FUNCTION_BLOCK EM_LiftingTransport EXTENDS EM_Base IMPLEMENTS I_EM_LiftingTransport

VAR_INPUT
//Inputs
	i_ref_stSettings : REFERENCE TO ST_SettingsLiftingTransport;
	
	// External interlocks (from outside this EM)
	i_fbExtIlckLiftUp : FB_Interlock;
	i_fbExtIlckLiftDown : FB_Interlock;
	i_fbExtIlckTransportExtract : FB_Interlock;
	i_fbExtIlckTransportRetract : FB_Interlock;
	
	i_refTB : REFERENCE TO OBJ_Carrier;	//Mogelijk voor uiteindelijke machine, voor de FUMO's is dit nog niet echt relevant
	
	i_eCtrlState		: E_CtrlState;
	
	s_arr_bTest : ARRAY[0..15] OF BOOL; 
END_VAR

VAR_OUTPUT
	q_bStaWarning : BOOL;
END_VAR

VAR

	//Interlocks	
	fbIlckHandlerLiftUp : FB_InterlockHandler;
	fbIlckHandlerLiftDown : FB_InterlockHandler;

	fbIlckHandlerTransportExtract : FB_InterlockHandler;
	fbIlckHandlerTransportRetract : FB_InterlockHandler;

//------------------------------------------//
	//Control Modules (Devices)
	axisLift : AXIS_REF;
	s_cmLift : CM_AX5000; // Including 2 limit switched and 1 reference switch

	axisTransport : AXIS_REF;
	s_cmTransport : CM_AX5000; // Including 2 limit switched and 1 reference switch
	
//------------------------------------------//

//------------------------------------------//
//Inputs
	s_diStaTrolleyOnPositionLeft : FB_DigInput;
	s_diStaTrolleyOnPositionRight : FB_DigInput;
	s_diStaCabinAreaOccupied : FB_DigInput;
	s_diStaCollisionAvoidanceSensor : FB_DigInput;
	s_diStaTrolleyLocked : FB_DigInput;
	s_diStaTrolleyUnlocked : FB_DigInput;
//------------------------------------------//	
	
//------------------------------------------//
//Outputs

//------------------------------------------//

	//Requests
	s_bReqGoToIdle : BOOL := FALSE;
	s_bReqPickTrolleyFromTB : BOOL := FALSE;
	s_bReqPlaceTrolleyInTB : BOOL := FALSE;

	//States
	s_bStaLiftDriveError : BOOL := FALSE;
	s_bStaTransportDriveError : BOOL := FALSE;
	
	s_bStaTrolleyInCabin : BOOL := FALSE;
	s_bStaTrolleyInTB : BOOL := FALSE;
		
	s_bStaTrolleyOnPositionLeft : BOOL := FALSE;
	s_bStaTrolleyOnPositionRight : BOOL := FALSE;
	s_bStaCabinAreaOccupied : BOOL := FALSE;
	s_bStaCollisionAvoidanceSensor : BOOL := FALSE;
	s_bStaTrolleyLocked : BOOL := FALSE;
	s_bStaTrolleyUnlocked : BOOL := FALSE;
	
	//Properties
	s_bStaAtIdlePosition : BOOL := FALSE;
	s_bStaTrolleyPickedFromTB : BOOL := FALSE;
	s_bStaTrolleyPlacedInTB : BOOL := FALSE;	

	//Interlockes	
	s_bIlckLiftUp : BOOL := TRUE;
	s_bIlckLiftDown : BOOL := TRUE;
	s_bIlckTransportExtract : BOOL := TRUE;
	s_bIlckTransportRetract : BOOL := TRUE;
	
//Alarms
	s_sReason : STRING;
	
	s_fbAlarmHandlerLiftDrive : FB_AlarmHandler;
	s_fbAlarmHandlerTransportDrive : FB_AlarmHandler;
	
	s_bErrLiftDrive : BOOL;
	s_bErrTransportDrive : BOOL;
	
	//Warnings
	s_fbAlarmHandlerSafetyDoorNotClosed : FB_AlarmHandler;
	s_bWrnSafetyDoorNotClosed : BOOL;
	
	s_bStaWarning : BOOL;
	
	s_sMessage : STRING;

	//Sequencers
	s_eSeqLiftingTransport : E_SeqLiftingTransport;
	s_fbSeqLiftingTransportControl : FB_SeqControl;

	s_eTmpLocation : E_Location;
	s_eTmpCenteringDone : BOOL;
	
	s_tMaxTravelTime : TIME;
	s_tDoorCheckTime : TIME;
	s_bDoorCheckTimeDisabled : BOOL := FALSE;
	

	//Hmi
	//Buttons
	s_fbHmiBtnGoToIdle					: FB_HmiBtn;
	s_fbHmiBtnPickTrolleyFromTB			: FB_HmiBtn;
	s_fbHmiBtnPlaceTrolleyInTB			: FB_HmiBtn;
		
	//Leds
	s_fbHmiLedTrolleyOnPositionLeft		: FB_HmiLed;
	s_fbHmiLedTrolleyOnPositionRight	: FB_HmiLed;
	s_fbHmiLedCabinAreaOccupied			: FB_HmiLed;
	s_fbHmiLedCollisionAvoidanceSensor	: FB_HmiLed;
	s_fbHmiLedTrolleyLocked				: FB_HmiLed;
	s_fbHmiLedTrolleyUnlocked			: FB_HmiLed;
	
	{warning '#TODO' Het zou beter zijn om dit onder te brengen in de onderstaande control modules}
	s_bHmiForceOutputEnabled : BOOL;
END_VAR

	
SUPER^();

METHOD PROTECTED _m_Alarms : BOOL

IF NOT SUPER^._m_Alarms() THEN
	RETURN;
END_IF

// Alarm Handlers
s_fbAlarmHandlerLiftDrive(
	i_bStaActive := s_bErrLiftDrive, 
	i_eAlarmLevel := E_AlarmLevel.Alarm, 
	i_sAlarmText := CONCAT(i_sEmName, CONCAT( ': Scissor Lift Drive error: ', s_sReason)));
	
s_fbAlarmHandlerTransportDrive(
	i_bStaActive := s_bErrTransportDrive, 
	i_eAlarmLevel := E_AlarmLevel.Alarm, 
	i_sAlarmText := CONCAT(i_sEmName, CONCAT( ': Transport Unit Drive error: ', s_sReason)));

// Reset warnings
IF i_bCmdReset THEN
	s_bWrnSafetyDoorNotClosed := FALSE;
END_IF

s_bStaError := 
	s_cmLift.p_bError
	OR s_cmTransport.p_bError
	OR s_fbAlarmHandlerLiftDrive.q_bStaActive
	OR s_fbAlarmHandlerTransportDrive.q_bStaActive;
	
s_bStaWarning :=
	s_fbAlarmHandlerSafetyDoorNotClosed.q_bStaActive;
	
_m_Alarms := TRUE;
END_METHOD

METHOD PRIVATE _m_AutomaticControl : BOOL

//Lifting Transport
_m_SeqLiftingTransport();
END_METHOD

METHOD PROTECTED _m_Devices : BOOL

IF NOT SUPER^._m_Devices() THEN
	RETURN;
END_IF

s_cmLift(
	i_bReqEnable := i_bReqEnable,
	i_eCtrlMode := i_eCtrlMode,
	i_bCmdReset := i_bCmdReset,
	i_refAxis := axisLift,
	i_bIclkForward := s_bIlckLiftUp,
	i_bIclkBackward := s_bIlckLiftDown);

s_bStaLiftDriveError := s_cmLift.p_bError;
	
s_cmTransport(
	i_bReqEnable := i_bReqEnable,
	i_eCtrlMode := i_eCtrlMode,
	i_bCmdReset := i_bCmdReset,
	i_refAxis := axisTransport,
	i_bIclkForward := s_bIlckTransportExtract, 
	i_bIclkBackward := s_bIlckTransportRetract);

s_bStaTransportDriveError := s_cmTransport.p_bError;

s_diStaTrolleyOnPositionLeft();
s_diStaTrolleyOnPositionRight();
s_diStaCabinAreaOccupied();
s_diStaCollisionAvoidanceSensor();
s_diStaTrolleyLocked();
s_diStaTrolleyUnlocked();

s_bStaTrolleyOnPositionLeft := s_diStaTrolleyOnPositionLeft.p_bStaInputDelayed;
s_bStaTrolleyOnPositionRight := s_diStaTrolleyOnPositionRight.p_bStaInputDelayed;
s_bStaCabinAreaOccupied := s_diStaCabinAreaOccupied.p_bStaInputDelayed;
s_bStaCollisionAvoidanceSensor := s_diStaCollisionAvoidanceSensor.p_bStaInputDelayed;
s_bStaTrolleyLocked := s_diStaTrolleyLocked.p_bStaInputDelayed;
s_bStaTrolleyUnlocked := s_diStaTrolleyUnlocked.p_bStaInputDelayed;

_m_Devices := TRUE;
END_METHOD

METHOD PROTECTED _m_Hmi : BOOL

IF NOT SUPER^._m_Hmi() THEN
	RETURN;
END_IF

//Buttons
s_fbHmiBtnGoToIdle();
s_fbHmiBtnPickTrolleyFromTB();
s_fbHmiBtnPlaceTrolleyInTB();

//Leds

s_fbHmiLedTrolleyOnPositionLeft(i_bStaLed := s_bStaTrolleyOnPositionLeft);
s_fbHmiLedTrolleyOnPositionRight(i_bStaLed := s_bStaTrolleyOnPositionRight);
s_fbHmiLedCabinAreaOccupied(i_bStaLed := s_bStaCabinAreaOccupied);
s_fbHmiLedCollisionAvoidanceSensor(i_bStaLed := s_bStaCollisionAvoidanceSensor);
s_fbHmiLedTrolleyLocked(i_bStaLed := s_bStaTrolleyLocked);
s_fbHmiLedTrolleyUnlocked(i_bStaLed := s_bStaTrolleyUnlocked);

_m_Hmi := TRUE;
END_METHOD

METHOD PROTECTED _m_Init : BOOL

IF NOT SUPER^._m_Init() THEN
	RETURN;
END_IF

//Control Modules
s_cmLift.i_bReqEnable := FALSE;
s_cmLift.i_eCtrlMode := E_CtrlMode.IDLE;
s_cmLift.i_sCmName := 'CM Lift';
s_cmLift.i_refAxis REF= axisLift;

s_cmTransport.i_bReqEnable := FALSE;
s_cmTransport.i_eCtrlMode := E_CtrlMode.IDLE;
s_cmTransport.i_sCmName := 'CM Transport Unit';
s_cmTransport.i_refAxis REF= axisTransport;
{warning '#TODO: Dot we need to added configuration parameters? Seperate struct or via settings or dedicateed variables'}

s_diStaTrolleyOnPositionLeft.i_stSettings.tmInputDelay := T#100MS;
s_diStaTrolleyOnPositionRight.i_stSettings.tmInputDelay := T#100MS;
s_diStaCabinAreaOccupied.i_stSettings.tmInputDelay := T#100MS;
s_diStaCollisionAvoidanceSensor.i_stSettings.tmInputDelay := T#100MS;
s_diStaTrolleyLocked.i_stSettings.tmInputDelay := T#100MS;
s_diStaTrolleyUnlocked.i_stSettings.tmInputDelay := T#100MS;

//Interlock strings
//Lift
//	i_stInterlockList.arr_Interlocks[0].sReason --> External, dynamical will be written in m_input
	fbIlckHandlerLiftDown.i_stInterlockList.arr_Interlocks[1].sReason := 'Transport not retracted';
//..fbIlckHandlerLiftDown.i_stInterlockList.arr_Interlocks[2].sReason := 'Transport not retracted';

//	i_stInterlockList.arr_Interlocks[0].sReason --> External, dynamical will be written in m_input
	fbIlckHandlerLiftUp.i_stInterlockList.arr_Interlocks[1].sReason := 'Trolly at correct position';
//..fbIlckHandlerLiftUp.i_stInterlockList.arr_Interlocks[2].sReason := '..';

//Transport
//	i_stInterlockList.arr_Interlocks[0].sReason --> External, dynamical will be written in m_input
	fbIlckHandlerTransportRetract.i_stInterlockList.arr_Interlocks[1].sReason := 'Lift not at correct position';
//..fbInterlockHandlerTransportRetract.i_stInterlockList.arr_Interlocks[2].sReason := 'Transport not retracted';

//	i_stInterlockList.arr_Interlocks[0].sReason --> External, dynamical will be written in m_input
	fbIlckHandlerTransportExtract.i_stInterlockList.arr_Interlocks[1].sReason := 'Lift not at correct position';
//..fbInterlockHandlerTransportExtract.i_stInterlockList.arr_Interlocks[2].sReason := '..';

//Hmi
	s_fbHmiBtnGoToIdle.p_eButtontype := E_HmiButtonType.PUSHBUTTON;
	s_fbHmiBtnGoToIdle.p_bStaVisible := FALSE;
	s_fbHmiBtnGoToIdle.p_bStaEnabled := FALSE;		
	s_fbHmiBtnGoToIdle.p_sBtnText := 'Go To Idle';
	
	s_fbHmiBtnPickTrolleyFromTB.p_eButtontype := E_HmiButtonType.PUSHBUTTON;
	s_fbHmiBtnPickTrolleyFromTB.p_bStaVisible := FALSE;
	s_fbHmiBtnPickTrolleyFromTB.p_bStaEnabled := FALSE;		
	s_fbHmiBtnPickTrolleyFromTB.p_sBtnText := 'Pick Trolley From TB';
	
	s_fbHmiBtnPlaceTrolleyInTB.p_eButtontype := E_HmiButtonType.PUSHBUTTON;
	s_fbHmiBtnPlaceTrolleyInTB.p_bStaVisible := FALSE;
	s_fbHmiBtnPlaceTrolleyInTB.p_bStaEnabled := FALSE;		
	s_fbHmiBtnPlaceTrolleyInTB.p_sBtnText := 'Place Trlley In TB';
	
	s_fbHmiLedTrolleyLocked				: FB_HmiLed;
	s_fbHmiLedTrolleyUnlocked			: FB_HmiLed;

	s_fbHmiLedTrolleyOnPositionLeft.p_bStaVisible := FALSE;
	s_fbHmiLedTrolleyOnPositionLeft.p_sToHmiDescriptionLed := 'Trolley On Position Left';
	
	s_fbHmiLedTrolleyOnPositionRight.p_bStaVisible := FALSE;
	s_fbHmiLedTrolleyOnPositionRight.p_sToHmiDescriptionLed := 'Trolley On Position Right';
	
	s_fbHmiLedCabinAreaOccupied.p_bStaVisible := FALSE;
	s_fbHmiLedCabinAreaOccupied.p_sToHmiDescriptionLed := 'Cabin Area Occupied';
	
	s_fbHmiLedCollisionAvoidanceSensor.p_bStaVisible := FALSE;
	s_fbHmiLedCollisionAvoidanceSensor.p_sToHmiDescriptionLed := 'Collision Avoidance Sensor';
	
	s_fbHmiLedTrolleyLocked.p_bStaVisible := FALSE;
	s_fbHmiLedTrolleyLocked.p_sToHmiDescriptionLed := 'Trolley Locked';
	
	s_fbHmiLedTrolleyUnlocked.p_bStaVisible := FALSE;
	s_fbHmiLedTrolleyUnlocked.p_sToHmiDescriptionLed := 'Trolley Unlocked';
	
_m_Init := TRUE;
END_METHOD

METHOD PROTECTED _m_Inputs : BOOL

IF NOT SUPER^._m_Inputs() THEN
	RETURN;
END_IF

//Interlocks
//Lift
fbIlckHandlerLiftDown.i_stInterlockList.arr_Interlocks[0].bState := i_fbExtIlckLiftDown.p_bInterlocked;
fbIlckHandlerLiftDown.i_stInterlockList.arr_Interlocks[0].sReason := i_fbExtIlckLiftDown.p_sReason;
fbIlckHandlerLiftDown.i_stInterlockList.arr_Interlocks[1].bState := NOT(s_cmTransport.p_fPosition = 0); //TODO
fbIlckHandlerLiftDown();

fbIlckHandlerLiftUp.i_stInterlockList.arr_Interlocks[0].bState := i_fbExtIlckLiftUp.p_bInterlocked;
fbIlckHandlerLiftUp.i_stInterlockList.arr_Interlocks[0].sReason := i_fbExtIlckLiftUp.p_sReason;
fbIlckHandlerLiftUp.i_stInterlockList.arr_Interlocks[1].bState := NOT(s_cmTransport.p_fPosition = 0); //TODO
fbIlckHandlerLiftUp();

s_bIlckLiftDown := fbIlckHandlerLiftDown.p_bInterlocked;
s_bIlckLiftUp := fbIlckHandlerLiftUp.p_bInterlocked;

//Transport
fbIlckHandlerTransportRetract.i_stInterlockList.arr_Interlocks[0].bState := i_fbExtIlckTransportRetract.p_bInterlocked;
fbIlckHandlerTransportRetract.i_stInterlockList.arr_Interlocks[0].sReason := i_fbExtIlckTransportRetract.p_sReason;
fbIlckHandlerTransportRetract.i_stInterlockList.arr_Interlocks[1].bState := NOT(s_cmLift.p_fPosition = 0); //TODO
fbIlckHandlerTransportRetract();

fbIlckHandlerTransportExtract.i_stInterlockList.arr_Interlocks[0].bState := i_fbExtIlckTransportExtract.p_bInterlocked;
fbIlckHandlerTransportExtract.i_stInterlockList.arr_Interlocks[0].sReason := i_fbExtIlckTransportExtract.p_sReason;
fbIlckHandlerTransportExtract.i_stInterlockList.arr_Interlocks[1].bState := NOT(s_cmLift.p_fPosition = 0); //TODO
fbIlckHandlerTransportExtract();

s_bIlckTransportRetract := fbIlckHandlerTransportRetract.p_bInterlocked;
s_bIlckTransportExtract := fbIlckHandlerTransportExtract.p_bInterlocked;

//Reasons (own reason first: Cm->Em->Un)
//Lift
IF s_bIlckLiftDown THEN
	s_cmLift.p_sInterlockedReasonDown := fbIlckHandlerLiftDown.p_sReason;
ELSE
	s_cmLift.p_sInterlockedReasonDown := '-';
END_IF
	
IF s_bIlckLiftUp THEN
	s_cmLift.p_sInterlockedReasonUp := fbIlckHandlerLiftUp.p_sReason;
ELSE
	s_cmLift.p_sInterlockedReasonUp := '-';
END_IF

//Transport
IF s_bIlckTransportRetract THEN
	s_cmTransport.p_sInterlockedReasonRetract := fbIlckHandlerTransportRetract.p_sReason;
ELSE
	s_cmTransport.p_sInterlockedReasonRetract := '-';
END_IF
	
IF s_bIlckTransportExtract THEN
	s_cmTransport.p_sInterlockedReasonExtract := fbIlckHandlerTransportExtract.p_sReason;
ELSE
	s_cmTransport.p_sInterlockedReasonExtract := '-';
END_IF

{warning '#TODO: Something similar needs to be added for lifting transport'}
//TB States (only use data if a valid ID is pressent else use sensor states)
IF __ISVALIDREF(i_refTB) AND (i_refTB.p_nId > 0) THEN
//++	s_bStaAtIdlePosition := i_refTB.p_b..;
//++	s_bStaTrolleyInTB := i_refTB.p_b..;
	s_bStaTrolleyInCabin := i_refTB.p_b..;
	//..
 
//--	s_bStaTB_CenteringDone := i_refTB.p_bCenteringDone;
//--	s_bStaTB_AtInfeed := i_refTB.p_eActLocation = E_Location.INFEED;
//--	s_bStaTB_AtCentering := i_refTB.p_eActLocation = E_Location.CENTERING;
//--	s_bStaTB_AtDocking := i_refTB.p_eActLocation = E_Location.DOCKING;
ELSE
//--	s_bStaTB_CenteringDone := s_eTmpCenteringDone;
//--	s_bStaTB_AtInfeed := s_bStaAtInfeedRearPosition OR s_bStaAtInfeedFrontPosition;
//--	s_bStaTB_AtCentering := s_bStaAtCenteringPosition;
//--	s_bStaTB_AtDocking := s_bStaAtDockingPosition;	
END_IF

_m_Inputs := TRUE;
END_METHOD

METHOD PRIVATE _m_ManualControl : BOOL

// Manual control has been implemented into lower layer control modules
END_METHOD

METHOD _m_MoveAbsolute : BOOL
VAR_INPUT
	i_ref_axis : REFERENCE TO TC2_MC2.AXIS_REF;
	i_ref_stProfile : ST_PositioningProfile;
END_VAR

VAR_INST
	s_MC_MoveAbsolute : TC2_MC2.MC_MoveAbsolute;
END_VAR

IF NOT(__ISVALIDREF(i_ref_axis)) THEN
	// Message invalid reference
	RETURN;
END_IF

s_MC_MoveAbsolute(
	Axis := i_ref_axis,
	Execute := TRUE AND NOT(s_MC_MoveAbsolute.Busy OR s_MC_MoveAbsolute.Done OR s_MC_MoveAbsolute.Error),
	Position := i_ref_stProfile.fPosition,
	Velocity := i_ref_stProfile.fVelocity,
	Acceleration := i_ref_stProfile.fAcceleration,
	Deceleration := i_ref_stProfile.fDeceleration,
	Jerk := i_ref_stProfile.fJerk,
	BufferMode := TC2_MC2.MC_BufferMode.MC_Aborting,
	Options := ,
	Done => ,
	Busy => ,
	Active => ,
	CommandAborted => ,
	Error => ,
	ErrorID => );
	
_m_MoveAbsolute := s_MC_MoveAbsolute.Done;
END_METHOD

METHOD PROTECTED _m_Outputs : BOOL

IF NOT SUPER^._m_Outputs() THEN
	RETURN;
END_IF

q_bStaWarning := s_bStaWarning;

_m_Outputs := TRUE;
END_METHOD

METHOD PROTECTED _m_Params : BOOL

IF NOT SUPER^._m_Params() THEN
	RETURN;
END_IF

//Write to settings
{warning '#TODO: Check what nees to be added here, is it nessecary add a fbParam for each parameter?'}
	
//++i_ref_stSettings.fSpeedManual := s_fbParamSpeedManual.p_fValue;

//++i_ref_stSettings.stLiftSpeedProfileJogging :=
//++i_ref_stSettings.stLiftSpeedProfilePositioning := 
//++i_ref_stSettings. 

_m_Params := TRUE;
END_METHOD

METHOD PRIVATE _m_SeqLiftingTransport : BOOL

s_fbHmiBtnTB_ToInfeed.p_bStaVisible := TRUE;
//--s_fbHmiBtnTB_ToInfeed.p_bStaEnabled := TRUE;

s_fbHmiBtnTB_ToCentering.p_bStaVisible := TRUE;
//--s_fbHmiBtnTB_ToCentering.p_bStaEnabled := TRUE;

s_fbHmiBtnTB_ToDocking.p_bStaVisible := TRUE;
//--s_fbHmiBtnTB_ToDocking.p_bStaEnabled := TRUE;

s_fbSeqLiftingTransportControl(
	i_nSeqStep := s_eSeqLiftingTransport, 
	i_sStepName := TO_STRING(s_eSeqLiftingTransport), 
	i_bCmdReset := i_bCmdReset
					AND (s_eSeqLiftingTransport = E_SeqTransport.ERROR) // Only reset/resume sequencer from ERROR state
					AND NOT(s_cmLift.p_bStaError)
					AND NOT(s_cmTransport.p_bStaError)
					AND i_bReqEnable, 
	i_bStaError := s_bStaError OR NOT(i_bReqEnable) AND FALSE);
	
CASE s_eSeqLiftingTransport OF
	
	E_SeqLiftingTransport.IDLE:
		s_eTmpLocation := E_Location.UNKNOWN;
	
		
		
		s_eSeqLiftingTransport := E_SeqLiftingTransport.START;
		
	E_SeqLiftingTransport.START:
		//--IF s_fbSeqTransportControl.q_tmStepTime > T#1S THEN
		//--	s_eSeqTransport := E_SeqTransport.READY;
		//--END_IF
		
		IF s_fbSeqLiftingTransportControl.q_bStaEntry THEN
			;//--s_cmPalletConveyor.m_Stop();
		END_IF		
	
		//IF s_cmPalletConveyor.p_bStaMotorStopped AND_THEN NOT(s_cmPalletConveyor.p_bStaBrakeReleased) AND s_fbSeqTransportControl.q_tmStepTime > T#1S THEN
		//	s_eSeqLiftingTransport := E_SeqTransport.READY;
		//END_IF
		
		s_cmLift.m_MC_Power(
			i_bEnable := TRUE,
			i_bEnablePositive := TRUE,
			i_bEnableNegative := TRUE,
			i_fOverride := 100.0,
			i_eBufferMode := TC2_MC2.MC_BufferMode.MC_Aborting);
			
		s_cmTransport.m_MC_Power(
			i_bEnable := TRUE,
			i_bEnablePositive := TRUE,
			i_bEnableNegative := TRUE,
			i_fOverride := 100.0,
			i_eBufferMode := TC2_MC2.MC_BufferMode.MC_Aborting);
		
		IF s_arr_bTest[0] THEN
			s_arr_bTest[0] := FALSE;
			s_eSeqLiftingTransport := E_SeqLiftingTransport.LIFT_PRE_PICK_TROLLEY_IN_TB;
		END_IF
	
	E_SeqLiftingTransport.HOME_TRANSPORT:
		IF s_fbSeqLiftingTransportControl.q_bStaEntry THEN
			s_cmTransport.m_MC_Home(
				i_bExecute := TRUE,
				i_fPosition := 0.0,
				i_eHomingMode := Tc2_MC2.MC_HomingMode.MC_Direct,
				i_eBufferMode := Tc2_MC2.MC_BufferMode.MC_Aborting);
		END_IF
		
		IF s_cmTransport.p_bDone THEN
			s_eSeqLiftingTransport := E_SeqLiftingTransport.HOME_LIFT;
		ELSIF s_cmTransport.p_bError THEN
			s_eSeqLiftingTransport := E_SeqLiftingTransport.ERROR;
		ELSIF s_fbSeqLiftingTransportControl.q_tmStepTime > T#30S THEN
			s_eSeqLiftingTransport := E_SeqLiftingTransport.ERROR;
		END_IF	
	
	E_SeqLiftingTransport.HOME_LIFT:
		IF s_fbSeqLiftingTransportControl.q_bStaEntry THEN
			s_cmLift.m_MC_Home(
				i_bExecute := TRUE,
				i_fPosition := 0.0,
				i_eHomingMode := Tc2_MC2.MC_HomingMode.MC_Direct,
				i_eBufferMode := Tc2_MC2.MC_BufferMode.MC_Aborting);
		END_IF
		
		IF s_cmLift.p_bDone THEN
			s_eSeqLiftingTransport := E_SeqLiftingTransport.HOME_LIFT;
		ELSIF s_cmLift.p_bError THEN
			s_eSeqLiftingTransport := E_SeqLiftingTransport.ERROR;
		ELSIF s_fbSeqLiftingTransportControl.q_tmStepTime > T#30S THEN
			s_eSeqLiftingTransport := E_SeqLiftingTransport.ERROR;
		END_IF		
	
	E_SeqLiftingTransport.MOVE_TO_IDLE:
	
/// PICK TROLLEY IN TB /////////////////////////////////////////////////////////
	E_SeqLiftingTransport.LIFT_PRE_PICK_TROLLEY_IN_TB:
		IF _m_MoveAbsolute(	i_ref_AXIS := axisLift, i_ref_stProfile := i_ref_stSettings.arr_LiftPositioningProfile[1]) THEN
			s_eSeqLiftingTransport := E_SeqLiftingTransport.TRANSPORT_PRE_PICK_TROLLEY_IN_TB;
		END_IF
	
	E_SeqLiftingTransport.TRANSPORT_PRE_PICK_TROLLEY_IN_TB:
		IF _m_MoveAbsolute(	i_ref_AXIS := axisTransport, i_ref_stProfile := i_ref_stSettings.arr_TransportPositioningProfile[1]) THEN
			s_eSeqLiftingTransport := E_SeqLiftingTransport.TRANSPORT_PICK_TROLLEY_IN_TB;
		END_IF
	
	E_SeqLiftingTransport.TRANSPORT_PICK_TROLLEY_IN_TB:
		IF _m_MoveAbsolute(	i_ref_AXIS := axisTransport, i_ref_stProfile := i_ref_stSettings.arr_TransportPositioningProfile[2]) THEN
			s_eSeqLiftingTransport := E_SeqLiftingTransport.LIFT_PICK_TROLLEY_IN_TB;
		END_IF
	
	E_SeqLiftingTransport.LIFT_PICK_TROLLEY_IN_TB:
		IF _m_MoveAbsolute(	i_ref_AXIS := axisLift, i_ref_stProfile := i_ref_stSettings.arr_LiftPositioningProfile[2]) THEN
			s_eSeqLiftingTransport := E_SeqLiftingTransport.LIFT_RAISE_TROLLEY_IN_TB;
		END_IF
	
	E_SeqLiftingTransport.LIFT_RAISE_TROLLEY_IN_TB:
		IF _m_MoveAbsolute(	i_ref_AXIS := axisLift, i_ref_stProfile := i_ref_stSettings.arr_LiftPositioningProfile[3]) THEN
			s_eSeqLiftingTransport := E_SeqLiftingTransport.TRANSPORT_PLACE_TROLLEY_IN_CABIN;
		END_IF

/// PLACE TROLLEY IN TB ////////////////////////////////////////////////////////	
	E_SeqLiftingTransport.TRANSPORT_PLACE_TROLLEY_IN_CABIN:
		IF _m_MoveAbsolute(	i_ref_AXIS := axisTransport, i_ref_stProfile := i_ref_stSettings.arr_TransportPositioningProfile[3]) THEN
			s_eSeqLiftingTransport := E_SeqLiftingTransport.LIFT_PRE_PLACE_TROLLEY_IN_CABIN;
		END_IF
		
	E_SeqLiftingTransport.LIFT_PRE_PLACE_TROLLEY_IN_CABIN:
		IF _m_MoveAbsolute(	i_ref_AXIS := axisLift, i_ref_stProfile := i_ref_stSettings.arr_LiftPositioningProfile[4]) THEN
			s_eSeqLiftingTransport := E_SeqLiftingTransport.LIFT_PLACE_TROLLEY_IN_CABIN;
		END_IF
		
	E_SeqLiftingTransport.LIFT_PLACE_TROLLEY_IN_CABIN:
		IF _m_MoveAbsolute(	i_ref_AXIS := axisLift, i_ref_stProfile := i_ref_stSettings.arr_LiftPositioningProfile[5]) THEN
			s_eSeqLiftingTransport := E_SeqLiftingTransport.LIFT_PRE_PICK_TROLLEY_IN_CABIN;
		END_IF

/// PICK TROLLEY IN CABIN //////////////////////////////////////////////////////		
	E_SeqLiftingTransport.LIFT_PRE_PICK_TROLLEY_IN_CABIN:
		IF _m_MoveAbsolute(	i_ref_AXIS := axisLift, i_ref_stProfile := i_ref_stSettings.arr_LiftPositioningProfile[6]) THEN
			s_eSeqLiftingTransport := E_SeqLiftingTransport.LIFT_PICK_TROLLEY_IN_CABIN;
		END_IF
		
	E_SeqLiftingTransport.LIFT_PICK_TROLLEY_IN_CABIN:
		IF _m_MoveAbsolute(	i_ref_AXIS := axisLift, i_ref_stProfile := i_ref_stSettings.arr_LiftPositioningProfile[7]) THEN
			s_eSeqLiftingTransport := E_SeqLiftingTransport.LIFT_RAISE_TROLLEY_IN_CABIN;
		END_IF
		
	E_SeqLiftingTransport.LIFT_RAISE_TROLLEY_IN_CABIN:
		IF _m_MoveAbsolute(	i_ref_AXIS := axisLift, i_ref_stProfile := i_ref_stSettings.arr_LiftPositioningProfile[8]) THEN
			s_eSeqLiftingTransport := E_SeqLiftingTransport.TRANSPORT_PRE_PLACE_TROLLEY_IN_TB;
		END_IF
	
/// PLACE TROLLEY IN TB //??////////////////////////////////////////////////////
	E_SeqLiftingTransport.TRANSPORT_PRE_PLACE_TROLLEY_IN_TB:
		IF _m_MoveAbsolute(	i_ref_AXIS := axisTransport, i_ref_stProfile := i_ref_stSettings.arr_TransportPositioningProfile[4]) THEN
			s_eSeqLiftingTransport := E_SeqLiftingTransport.TRANSPORT_PLACE_TROLLEY_IN_TB;
		END_IF
	
	E_SeqLiftingTransport.TRANSPORT_PLACE_TROLLEY_IN_TB:
		IF _m_MoveAbsolute(	i_ref_AXIS := axisTransport, i_ref_stProfile := i_ref_stSettings.arr_TransportPositioningProfile[5]) THEN
			s_eSeqLiftingTransport := E_SeqLiftingTransport.LIFT_PRE_PLACE_TROLLEY_IN_TB;
		END_IF

	E_SeqLiftingTransport.LIFT_PRE_PLACE_TROLLEY_IN_TB:
		IF _m_MoveAbsolute(	i_ref_AXIS := axisLift, i_ref_stProfile := i_ref_stSettings.arr_LiftPositioningProfile[9]) THEN
			s_eSeqLiftingTransport := E_SeqLiftingTransport.LIFT_PLACE_TROLLEY_IN_TB;
		END_IF
		
	E_SeqLiftingTransport.LIFT_PLACE_TROLLEY_IN_TB:
		IF _m_MoveAbsolute(	i_ref_AXIS := axisLift, i_ref_stProfile := i_ref_stSettings.arr_LiftPositioningProfile[10]) THEN
			s_eSeqLiftingTransport := E_SeqLiftingTransport.START;
		END_IF
		
	E_SeqLiftingTransport.READY:
		IF s_fbSeqLiftingTransportControl.q_bStaEntry THEN
			i_refTB.p_eLocation := s_eTmpLocation;
			s_eTmpLocation := E_Location.UNKNOWN;
		END_IF
		
(*		i_refTB.p_bOuterDoorOpened S= s_bStaAtInfeedRearPosition AND s_bStaAtInfeedFrontPosition AND s_bStaDoorOpened;
	
		IF s_fbHmiBtnTB_ToInfeed.p_osrBtnPress OR s_bReqTB_ToInfeed THEN
			IF m_CmdTB_ToInfeed(o_sReason => s_sMessage) THEN
				s_eSeqTransport := E_SeqTransport.MOVE_TO_INFEED;
			ELSE	
				//Write message
				//--s_sMessage := m_TB_ToCenter.o_sReason;
			END_IF
 
			s_bReqTB_ToInfeed := FALSE;
			
			//--AND NOT(s_bStaAtInfeedRearPosition)
			//--THEN
			
		ELSIF s_fbHmiBtnTB_ToCentering.p_osrBtnPress OR s_bReqTB_ToCenter THEN
			IF m_CmdTB_ToCenter(o_sReason => s_sMessage) THEN
				s_eSeqTransport := E_SeqTransport.MOVE_TO_CENTERING;
			ELSE	
				//Write message
				//--s_sMessage := m_TB_ToCenter.o_sReason;
			END_IF	
		
			s_bReqTB_ToCenter := FALSE;
			
			//--AND NOT(s_bStaAtCenteringPosition)
			//--THEN
			
			//--IF s_bStaDoorOpened THEN
			//--	s_eSeqTransport := E_SeqTransport.MOVE_TO_Centering;
			//--ELSE
			//--	s_bWrnOuterDoorNotOpened := TRUE;
			//--END_IF
			
		ELSIF s_fbHmiBtnTB_ToDocking.p_osrBtnPress OR s_bReqTB_ToDocking THEN
			IF m_CmdTB_ToDocking(o_sReason => s_sMessage) THEN
				s_eSeqTransport := E_SeqTransport.MOVE_TO_DOCKING;
			ELSE	
				//Write message
				//--s_sMessage := m_TB_ToDocking.o_sReason;
			END_IF	
		
			s_bReqTB_ToDocking := FALSE;
			
		//--	AND NOT(s_bStaAtDockingPosition)
		//--	THEN
		//--	s_eSeqTransport := E_SeqTransport.MOVE_TO_DOCKING;
		END_IF	
	
	E_SeqTransport.MOVE_TO_INFEED:
		IF s_fbSeqTransportControl.q_bStaEntry THEN		
			s_tMaxTravelTime := LREAL_TO_TIME((i_ref_stSettings.fDistanceToInfeed / i_ref_stSettings.fSpeedGoToInfeed) * i_ref_stSettings.fTravelTollerance * 1000);
			s_cmPalletConveyor.m_StartBackward(i_rTargetSpeed := i_stSettings.fSpeedGoToInfeed);
		END_IF
		
		IF s_bStaAtInfeedRearPosition THEN
			s_eTmpLocation := E_Location.INFEED;
			s_eSeqTransport := E_SeqTransport.STOP;
		ELSIF s_fbSeqTransportControl.q_tmStepTime > s_tMaxTravelTime THEN
			s_bErrTravelTimeOut := TRUE;
			s_sReason := 'Moving to infeed - timeout';
			s_eSeqTransport := E_SeqTransport.ERROR;
		END_IF
	
	E_SeqTransport.MOVE_TO_CENTERING:
		IF s_fbSeqTransportControl.q_bStaEntry THEN
			s_tMaxTravelTime := LREAL_TO_TIME((i_ref_stSettings.fDistanceToCentering / i_ref_stSettings.fSpeedGoToCentering) * i_ref_stSettings.fTravelTollerance * 1000);
			s_tDoorCheckTime := LREAL_TO_TIME((i_ref_stSettings.fDistanceOuteDoorCheck / i_ref_stSettings.fSpeedGoToCentering) * 1000);
			s_cmPalletConveyor.m_StartForward(i_rTargetSpeed := i_stSettings.fSpeedGoToCentering);
		END_IF
		
		IF s_bStaAtCenteringPosition THEN
			s_bDoorCheckTimeDisabled := FALSE;
			s_eTmpLocation := E_Location.CENTERING;
			s_eSeqTransport := E_SeqTransport.STOP;
		
		ELSIF s_fbSeqTransportControl.q_tmStepTime < s_tDoorCheckTime 
			AND NOT(s_bStaDoorOpened) THEN
			s_bWrnOuterDoorNotOpened := TRUE;
			s_bDoorCheckTimeDisabled := TRUE; //Disable error after first occurance (to prevent invalid retriggering at reties)
			s_eSeqTransport := E_SeqTransport.ERROR;
			
		ELSIF s_fbSeqTransportControl.q_tmStepTime > s_tMaxTravelTime THEN
			s_bErrTravelTimeOut := TRUE;
			s_sReason := 'Moving to Centering - timeout';
			s_eSeqTransport := E_SeqTransport.ERROR;

		//--Not clear it this will work correct due to order of sensor positions
		//--ELSIF s_bStaAtDockingPosition THEN
		//--	s_bErrTravelTimeOut := TRUE;
		//--	s_sReason := 'Moving to Centering - too far (docking)';
		//--	s_eSeqTransport := E_SeqTransport.ERROR;
		
		END_IF
	
	E_SeqTransport.MOVE_TO_DOCKING:
		IF s_fbSeqTransportControl.q_bStaEntry THEN
			s_tMaxTravelTime := LREAL_TO_TIME((i_ref_stSettings.fDistanceToDocking / i_ref_stSettings.fSpeedGoToDocking) * i_ref_stSettings.fTravelTollerance * 1000);
			s_cmPalletConveyor.m_StartForward(i_rTargetSpeed := i_stSettings.fSpeedGoToDocking);
		END_IF
		
		IF s_bStaAtDockingPosition THEN
			s_eTmpLocation := E_Location.DOCKING;
			s_eSeqTransport := E_SeqTransport.STOP;
		ELSIF s_fbSeqTransportControl.q_tmStepTime > s_tMaxTravelTime THEN
			s_bErrTravelTimeOut := TRUE;
			s_sReason := 'Moving to docking - timeout';
			s_eSeqTransport := E_SeqTransport.ERROR;		
		END_IF
		
	E_SeqTransport.STOP:
		IF s_fbSeqTransportControl.q_bStaEntry THEN
			s_cmPalletConveyor.m_Stop();
		END_IF
		
		IF s_cmPalletConveyor.p_bStaMotorStopped THEN
			s_eSeqTransport := E_SeqTransport.READY;
		END_IF
		
	E_SeqTransport.ERROR:
		s_cmPalletConveyor.m_Stop();
*)		
END_CASE
END_METHOD

METHOD PUBLIC m_CmdCenteringTB : BOOL
VAR_INPUT
	i_refReason : REFERENCE TO STRING;
END_VAR
VAR_OUTPUT
	o_sReason : STRING;
END_VAR

IF NOT i_bReqEnable THEN 
	RETURN;
END_IF

//--IF NOT(s_bIlckCenteringToCenter) THEN
//--	s_bReqCenteringTB := TRUE;
//--	m_CenteringTB := TRUE;
//--ELSE
//--	m_CenteringTB := FALSE;	
//--END_IF

IF s_bIlckCenteringToCenter THEN
	i_refReason := 'Command Centering: Interlocked';
	m_CmdCenteringTB := FALSE;
ELSE
	m_CmdCenteringTB := TRUE;	
END_IF
END_METHOD

METHOD PUBLIC m_CmdTB_ToCenter : BOOL
VAR_OUTPUT
	o_sReason : STRING;
END_VAR

IF NOT i_bReqEnable THEN 
	RETURN;
END_IF

//--IF NOT(s_bIlckConveyorForward) 
//--	AND NOT(s_bStaAtCenteringPosition)
//--	THEN
//--	s_bReqTB_ToCenter := TRUE;
//--	m_TB_ToCenter := TRUE;
//--ELSE
//--	m_TB_ToCenter := FALSE;	
//--END_IF

////////

IF s_bIlckConveyorForward THEN
	o_sReason := 'Command To Center: Interlocked';
	m_CmdTB_ToCenter := FALSE;
ELSIF s_bStaAtCenteringPosition THEN
 	o_sReason := 'Already at center position';
	m_CmdTB_ToCenter := FALSE;
ELSIF NOT(s_bStaDoorOpened) THEN
	o_sReason := 'Door not opened';
	s_bWrnOuterDoorNotOpened := TRUE; // kan mogelijk vervallen wanneer er toch gewerkt gaat worden met reasons.
	m_CmdTB_ToCenter := FALSE;
ELSE
	m_CmdTB_ToCenter := TRUE;	
END_IF
END_METHOD

METHOD PUBLIC m_CmdTB_ToDocking : BOOL
VAR_OUTPUT
	o_sReason : STRING;
END_VAR

IF NOT i_bReqEnable THEN 
	RETURN;
END_IF

//--IF NOT(s_bIlckConveyorForward) THEN
//--	s_bReqTB_ToDocking := TRUE;
//--	m_TB_ToDocking := TRUE;
//--ELSE
//--	m_TB_ToDocking := FALSE;	
//--END_IF

IF s_bStaAtDockingPosition THEN
	o_sReason := 'Command to Docking: Interlocked';
	m_CmdTB_ToDocking := FALSE;
ELSE
	m_CmdTB_ToDocking := TRUE;	
END_IF
END_METHOD

METHOD PUBLIC m_CmdTB_ToInfeed : BOOL
VAR_OUTPUT
	o_sReason : STRING;
END_VAR

IF NOT i_bReqEnable THEN 
	RETURN;
END_IF

//--IF NOT(s_bIlckConveyorBackward) 
//--	AND NOT(s_bStaAtInfeedRearPosition)
//--	THEN
//--	s_bReqTB_ToInfeed := TRUE;
//--	m_TB_ToInfeed := TRUE;
//--ELSE
//--	m_TB_ToInfeed := FALSE;	
//--END_IF

IF s_bIlckConveyorBackward THEN
	o_sReason := 'Command to Infeed: Interlocked';
	m_CmdTB_ToInfeed := FALSE;
ELSE
	m_CmdTB_ToInfeed := TRUE;	
END_IF
END_METHOD

METHOD PUBLIC m_Main : BOOL

IF NOT SUPER^.m_Main() THEN
	RETURN;
END_IF

CASE i_eCtrlMode OF

	E_CtrlMode.IDLE:
		s_eSeqLiftingTransport := E_SeqLiftingTransport.IDLE;
		
	E_CtrlMode.AUTOMATIC:
		//Automatic commands are controlled by higher-layer unit
		_m_AutomaticControl();
		
	E_CtrlMode.MANUAL:
		//Execute manaual control (based on HMI buttons)
		
		//Manual commands (convert HMI buttons to requests), only in state running
		IF (i_eCtrlState = E_CtrlState.RUNNING) THEN
			s_bReqGoToIdle := s_fbHmiBtnGoToIdle.p_osrBtnPress;
			s_bReqPickTrolleyFromTB := s_fbHmiBtnPickTrolleyFromTB.p_osrBtnPress;
			s_bReqPlaceTrolleyInTB := s_fbHmiBtnPlaceTrolleyInTB.p_osrBtnPress;
		END_IF
	
		_m_AutomaticControl();
		
	E_CtrlMode.MAINTENANCE:
		//Execute maintenance control (HMI control module buttons)
		//Reset automatic/manual sequencer
		s_eSeqLiftingTransport := E_SeqTransport.IDLE;
	
		; 	//Maintenance control is implemented in lower-layer control modules
	
	E_CtrlMode.IO:
		//Execute IO-test control (HMI output force control)
		; 	//IO-Test control is implemented in lower-layer control modules
			//Enabling control is done direcly under this case instruction
		
	E_CtrlMode.CLEANING:
		//Execute cleaning control (cleaning  specific functionalities)
		;	//Cleaning control is not implemented, this could be a done in the future if neccesary
				
END_CASE

//AUTOMATIC-mode //////////////////////////////////////////////////////////////////////////////////

//MANUAL-mode /////////////////////////////////////////////////////////////////////////////////////

//Buttons visibility
IF (i_eCtrlMode = E_CtrlMode.MANUAL) THEN
	s_fbHmiBtnGoToIdle.p_bStaVisible := TRUE;
	s_fbHmiBtnPickTrolleyFromTB.p_bStaVisible := TRUE;
	s_fbHmiBtnPlaceTrolleyInTB.p_bStaVisible := TRUE;
ELSE
	s_fbHmiBtnGoToIdle.p_bStaVisible := FALSE;
	s_fbHmiBtnPickTrolleyFromTB.p_bStaVisible := FALSE;
	s_fbHmiBtnPlaceTrolleyInTB.p_bStaVisible := FALSE;
END_IF

//Buttons enabling
IF i_bReqEnable AND (i_eCtrlMode = E_CtrlMode.MANUAL) AND (i_eCtrlState = E_CtrlState.RUNNING) THEN

	//Lift/Transport
	s_fbHmiBtnGoToIdle.p_bStaEnabled :=
		NOT(s_bIlckLiftDown)
		AND NOT(s_bIlckLiftUp)
		AND NOT(s_bIlckTransportRetract)
		AND NOT(s_bIlckTransportExtract)
		AND NOT(s_cmLift.p_bStaError)
		AND NOT(s_cmTransport.p_bStaError);
	
	s_fbHmiBtnPickTrolleyFromTB.p_bStaEnabled :=
		NOT(s_bIlckLiftDown)
		AND NOT(s_bIlckLiftUp)
		AND NOT(s_bIlckTransportRetract)
		AND NOT(s_bIlckTransportExtract)
		AND NOT(s_cmLift.p_bStaError)
		AND NOT(s_cmTransport.p_bStaError);

	s_fbHmiBtnPlaceTrolleyInTB.p_bStaEnabled :=
		NOT(s_bIlckLiftDown)
		AND NOT(s_bIlckLiftUp)
		AND NOT(s_bIlckTransportRetract)
		AND NOT(s_bIlckTransportExtract)
		AND NOT(s_cmLift.p_bStaError)
		AND NOT(s_cmTransport.p_bStaError);	
		
ELSE
	s_fbHmiBtnGoToIdle.p_bStaEnabled := FALSE;
	s_fbHmiBtnPickTrolleyFromTB.p_bStaEnabled := FALSE;
	s_fbHmiBtnPlaceTrolleyInTB.p_bStaEnabled := FALSE;
END_IF

//MAINTENANCE-mode ////////////////////////////////////////////////////////////////////////////////

//Stopping control modules
IF (i_eCtrlMode = E_CtrlMode.MAINTENANCE) AND (i_eCtrlState = E_CtrlState.STOPPING) THEN 
	s_cmLift.m_MC_Stop(
		i_bExecute := TRUE,
		i_fDeceleration := i_ref_stSettings.stLiftSpeedProfilePositioning.fDeceleration,
		i_fJerk := i_ref_stSettings.stLiftSpeedProfilePositioning.fJerk);
		
	s_cmTransport.m_MC_Stop(
		i_bExecute := TRUE,
		i_fDeceleration := i_ref_stSettings.stTransportSpeedProfilePositioning.fDeceleration,
		i_fJerk := i_ref_stSettings.stTransportSpeedProfilePositioning.fJerk);
END_IF

//IO-mode /////////////////////////////////////////////////////////////////////////////////////////
IF (i_eCtrlMode = E_CtrlMode.IO) AND (i_eCtrlState = E_CtrlState.RUNNING) THEN
	s_bHmiForceOutputEnabled := TRUE;
ELSE
	s_bHmiForceOutputEnabled := FALSE;	
END_IF

m_Main := TRUE;
END_METHOD

{attribute 'TcRpcEnable'}
METHOD PUBLIC m_ReqCenteringTB : BOOL

IF NOT i_bReqEnable THEN 
	RETURN;
END_IF

IF NOT i_bReqEnable THEN 
	RETURN;
END_IF

s_bReqCenteringTB := TRUE;

m_ReqCenteringTB := TRUE;
END_METHOD

{attribute 'TcRpcEnable'}
METHOD PUBLIC m_ReqTB_ToCenter : BOOL

IF NOT i_bReqEnable THEN 
	RETURN;
END_IF

s_bReqTB_ToCenter := TRUE;

m_ReqTB_ToCenter := TRUE;
END_METHOD

{attribute 'TcRpcEnable'}
METHOD PUBLIC m_ReqTB_ToDocking : BOOL

IF NOT i_bReqEnable THEN 
	RETURN;
END_IF

s_bReqTB_ToDocking := TRUE;

m_ReqTB_ToDocking := TRUE;
END_METHOD

{attribute 'TcRpcEnable'}
METHOD PUBLIC m_ReqTB_ToInfeed : BOOL

IF NOT i_bReqEnable THEN 
	RETURN;
END_IF

s_bReqTB_ToInfeed := TRUE;

m_ReqTB_ToInfeed := TRUE;
END_METHOD

PROPERTY PUBLIC p_bStaTB_AtCentering : BOOL
GET

p_bStaTB_AtCentering := s_bStaTB_AtCentering;
END_GET
END_PROPERTY

PROPERTY PUBLIC p_bStaTB_AtDocking : BOOL
GET

p_bStaTB_AtDocking := s_bStaTB_AtDocking;
END_GET
END_PROPERTY

PROPERTY PUBLIC p_bStaTB_AtInfeed : BOOL
GET

p_bStaTB_AtInfeed := s_bStaTB_AtInfeed;
END_GET
END_PROPERTY

PROPERTY PUBLIC p_bStaTB_CenteringDone : BOOL
GET

p_bStaTB_CenteringDone := s_bStaTB_CenteringDone;
END_GET
END_PROPERTY

END_FUNCTION_BLOCK

(* stored: Version 1.1.0.1, ProductVersion 3.1.4024.12
   POU EM_LiftingTransport: Id {82ac1e56-2937-4df1-886d-5bc6dc15361f}, SpecialFunc None
   Folder Base: Id {aa880d32-2da2-45ff-bcea-b6be34b0a44b}
   Method _m_Alarms: Id {77ac2c1c-b354-4acb-9f0d-e0fd9e0a3a94}
   Method _m_AutomaticControl: Id {51dbf1d4-9c3c-42ad-87fe-cdadd1984100}
   Method _m_Devices: Id {b95b1090-f72e-49a8-b75a-87fbc22bb2f7}
   Method _m_Hmi: Id {86cd5a15-a053-432c-9e95-504bd0cfab5b}
   Method _m_Init: Id {fdcbf52e-0860-4b94-915e-8e7c2bbd0a27}
   Method _m_Inputs: Id {2c09f905-698a-4dfd-8c60-1a7d7f6d646b}
   Method _m_ManualControl: Id {61a84643-dbec-4bc1-99bd-3a2ec3342898}
   Method _m_MoveAbsolute: Id {7f8f7561-70c1-4897-9a57-d3b7b8c51729}
   Method _m_Outputs: Id {0027b51b-0e3b-4c47-b79c-c262d8cada1b}
   Method _m_Params: Id {5f8e46d4-1bd2-48a0-a796-5af6a0b2577f}
   Method _m_SeqLiftingTransport: Id {adfb5128-2b00-4a29-b7de-b50ba035879a}
   Method m_CmdCenteringTB: Id {5f07294c-c083-4786-a1a2-586c95e439f7}
   Method m_CmdTB_ToCenter: Id {3a534c15-c636-468b-8b82-6fd59e761d1a}
   Method m_CmdTB_ToDocking: Id {fddfe49e-6281-47a3-8534-8abf984608e2}
   Method m_CmdTB_ToInfeed: Id {05a177ec-65c8-4b07-91b0-bc7997926449}
   Method m_Main: Id {7d708d4c-1fee-4511-a8d0-db3dbe3fd7e6}
   Method m_ReqCenteringTB: Id {415ce6ea-afb8-4118-a1fc-ea58b530d7b6}
   Method m_ReqTB_ToCenter: Id {9d30bbef-bcd6-4fc2-8d93-9b2201ca737f}
   Method m_ReqTB_ToDocking: Id {bc26af41-4ec1-4049-ae2f-a8f4c7a26c9b}
   Method m_ReqTB_ToInfeed: Id {fa516528-012b-4031-8e18-317ece30b039}
   Property p_bStaTB_AtCentering: Id {050383f4-1821-4a98-ab50-f2e654340431}
   Get Get: Id {03f3f379-9c7e-473c-8407-742758c9f4b6}
   Property p_bStaTB_AtDocking: Id {630d4760-3c9e-490a-b1db-ceb84ce3b93d}
   Get Get: Id {ac0f1cfe-6ddb-4648-8ead-590b388c0171}
   Property p_bStaTB_AtInfeed: Id {ccba55b7-671b-48a2-af2d-7bdd569222c9}
   Get Get: Id {c55ed7dc-3eae-49e0-bba0-c67b4ed5fb10}
   Property p_bStaTB_CenteringDone: Id {92f12f64-9c7b-449f-90f0-528b8c0b82e0}
   Get Get: Id {f8e455bd-3d78-46ed-aec1-a530ae8bd329} *)
